{attribute 'qualified_only'}
{attribute 'strict'}
TYPE eGensetStartStop :
(
	Auto := 0,
	Stop := 1,
	Start := 2
);
END_TYPE

(* stored: Version 1.1.0.1, ProductVersion 3.1.4026.18
   DUT eGensetStartStop: Id {c733e097-8e3a-478a-9eca-23da55d9c024} *)
